TYPE ST_PhtcCtrl :
STRUCT
	bStopInfeedConveyor:BOOL;
	bStopSeparator:BOOL;
END_STRUCT
END_TYPE

(* stored: Version 1.1.0.1, ProductVersion 3.1.4024.15
   DUT ST_PhtcCtrl: Id {f01ae20b-dda9-422c-82b5-c017f17d27fd} *)
